FUNCTION F_ComputeInt32Size : UDINT
VAR_INPUT
    nValue  : DINT;
END_VAR


IF nValue >= 0 THEN
    F_ComputeInt32Size := F_ComputeRawVarint32Size(TO_UDINT(nValue));
ELSE
    // Must sign-extend.
    F_ComputeInt32Size := 10;    
END_IF

END_FUNCTION

(* stored: Version 1.1.0.1
   POU F_ComputeInt32Size: Id {88b0525d-445f-4b96-bae4-76ae8cc87be9}, SpecialFunc None *)
